(* Logix 5000 project; controller AdvManLab vendor 1 type 14 code 158 rev 28.12; software revision 28.01; part 12 of 13 *)
(* tags used below, declared in another part *)
   ABB_Loop_Conv_ES_Ch1 : BOOL;   // Cell 3 Conveyor Pull Cord / E-Stop Ch1
   ABB_Loop_Conv_ES_Ch2 : BOOL;   // Cell 3 Conveyor Pull Cord / E-Stop Ch2
   ABBLoopSTO_O1 : BOOL;
   ABBLoopSTO_O2 : BOOL;
   C1_Robot_ES_OK : BOOL;
   C1_Robot_Gates_OK : BOOL;
   C1EASRelay_Monitor : BOOL;   // Robot External Safety Gate Relay Monitor
   C1EESRelay_Monitor : BOOL;   // Robot External EStop Relay Monitor
   C1S : Fanuc_Cell_Safe;
   C2_Robot_ES_OK : BOOL;
   C2_Robot_Gates_OK : BOOL;
   C2EASRelay_Monitor : BOOL;   // Robot External Safety Gate Relay Monitor
   C2EESRelay_Monitor : BOOL;   // Robot External EStop Relay Monitor
   C2S : Fanuc_Cell_Safe;
   C3_Robot_ES_OK : BOOL;
   C3_Robot_Gates_OK : BOOL;
   C3EASRelay_Monitor : BOOL;   // Robot External Safety Gate Relay Monitor
   C3EESRelay_Monitor : BOOL;   // Robot External EStop Relay Monitor
   C3S : ABB_Cell_Safe;
   Cell_1 : Fanuc_Cell;
   Cell_2 : Fanuc_Cell;
   Fanuc_Loop_Conv_ES_Ch1 : BOOL;   // Cell 1/2 Conveyor Pull Cord / E-Stop Ch1
   Fanuc_Loop_Conv_ES_Ch2 : BOOL;   // Cell 1/2 Conveyor Pull Cord / E-Stop Ch2
   FanucLoopSTO_O1 : BOOL;
   FanucLoopSTO_O2 : BOOL;
   MainPnlESCH1 : BOOL;   // Main Panel E-Stop Button CH1
   MainPnlESCH2 : BOOL;   // Main Panel E-Stop Button CH2
   RungCommentS : BOOL;
   Unused_S_In : BOOL;   // Tag to indicate bit is unused in I/O mapping
   Unused_S_Out : BOOL;   // Unused Safety Output - Replace as needed
(* SafetyProgram, continued *)

ROUTINE MainRoutine   (* ladder *)
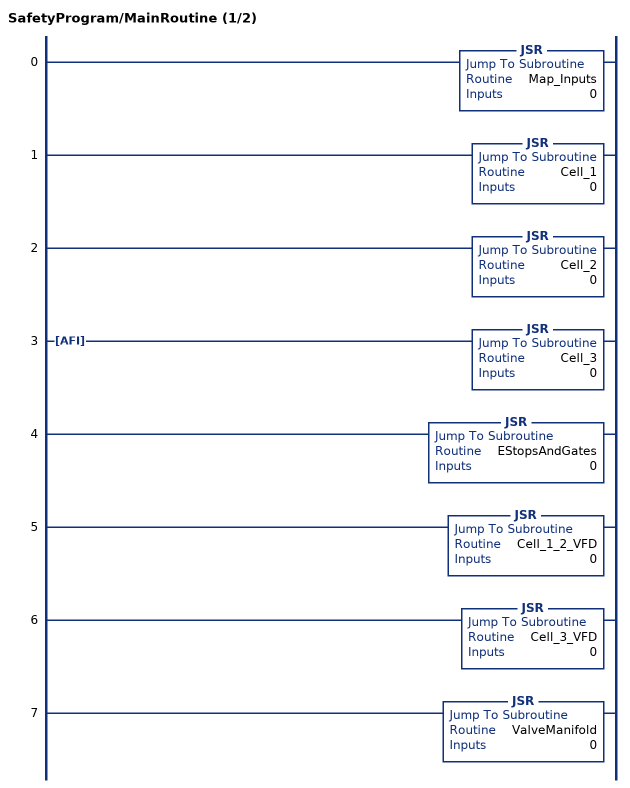
   0: JSR(Map_Inputs,0);
   1: JSR(Cell_1,0);
   2: JSR(Cell_2,0);
   3: AFI()JSR(Cell_3,0);
   4: JSR(EStopsAndGates,0);
   5: JSR(Cell_1_2_VFD,0);
   6: JSR(Cell_3_VFD,0);
   7: JSR(ValveManifold,0);
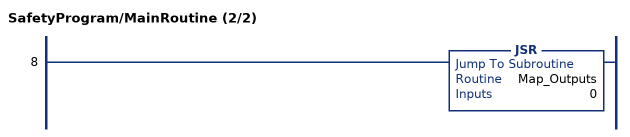
   8: JSR(Map_Outputs,0);
END_ROUTINE

ROUTINE Map_Inputs   (* ladder *)
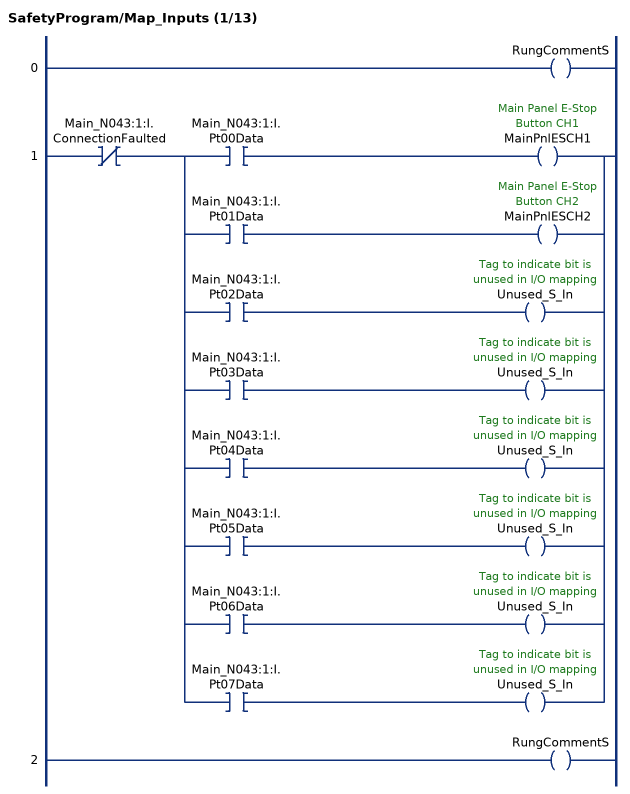
   0: OTE(RungCommentS);
   1: XIO(Main_N043:1:I.ConnectionFaulted)[XIC(Main_N043:1:I.Pt00Data) OTE(MainPnlESCH1) ,XIC(Main_N043:1:I.Pt01Data) OTE(MainPnlESCH2) ,XIC(Main_N043:1:I.Pt02Data) OTE(Unused_S_In) ,XIC(Main_N043:1:I.Pt03Data) OTE(Unused_S_In) ,XIC(Main_N043:1:I.Pt04Data) OTE(Unused_S_In) ,XIC(Main_N043:1:I.Pt05Data) OTE(Unused_S_In) ,XIC(Main_N043:1:I.Pt06Data) OTE(Unused_S_In) ,XIC(Main_N043:1:I.Pt07Data) OTE(Unused_S_In) ];
   2: OTE(RungCommentS);
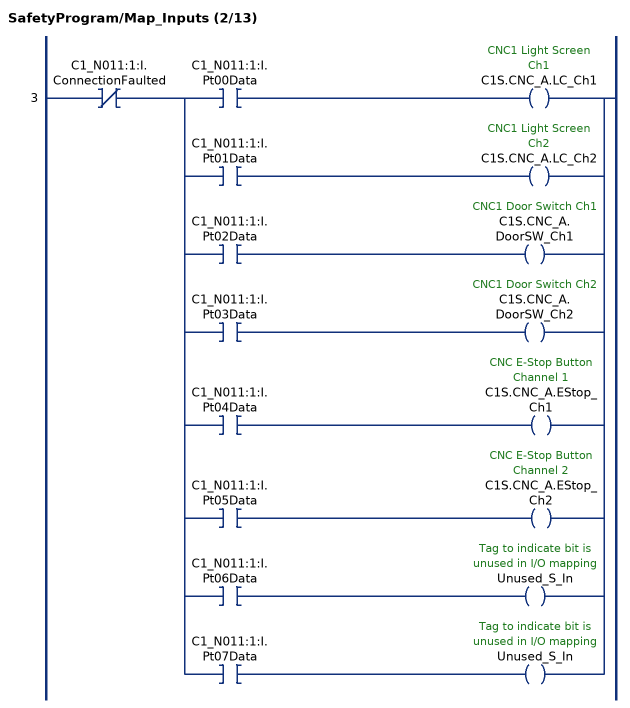
   3: XIO(C1_N011:1:I.ConnectionFaulted)[XIC(C1_N011:1:I.Pt00Data) OTE(C1S.CNC_A.LC_Ch1) ,XIC(C1_N011:1:I.Pt01Data) OTE(C1S.CNC_A.LC_Ch2) ,XIC(C1_N011:1:I.Pt02Data) OTE(C1S.CNC_A.DoorSW_Ch1) ,XIC(C1_N011:1:I.Pt03Data) OTE(C1S.CNC_A.DoorSW_Ch2) ,XIC(C1_N011:1:I.Pt04Data) OTE(C1S.CNC_A.EStop_Ch1) ,XIC(C1_N011:1:I.Pt05Data) OTE(C1S.CNC_A.EStop_Ch2) ,XIC(C1_N011:1:I.Pt06Data) OTE(Unused_S_In) ,XIC(C1_N011:1:I.Pt07Data) OTE(Unused_S_In) ];
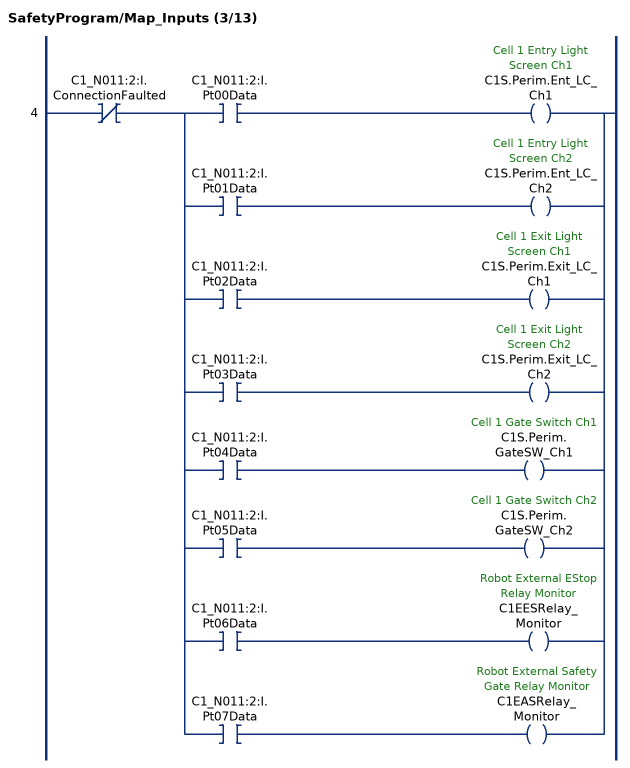
   4: XIO(C1_N011:2:I.ConnectionFaulted)[XIC(C1_N011:2:I.Pt00Data) OTE(C1S.Perim.Ent_LC_Ch1) ,XIC(C1_N011:2:I.Pt01Data) OTE(C1S.Perim.Ent_LC_Ch2) ,XIC(C1_N011:2:I.Pt02Data) OTE(C1S.Perim.Exit_LC_Ch1) ,XIC(C1_N011:2:I.Pt03Data) OTE(C1S.Perim.Exit_LC_Ch2) ,XIC(C1_N011:2:I.Pt04Data) OTE(C1S.Perim.GateSW_Ch1) ,XIC(C1_N011:2:I.Pt05Data) OTE(C1S.Perim.GateSW_Ch2) ,XIC(C1_N011:2:I.Pt06Data) OTE(C1EESRelay_Monitor) ,XIC(C1_N011:2:I.Pt07Data) OTE(C1EASRelay_Monitor) ];
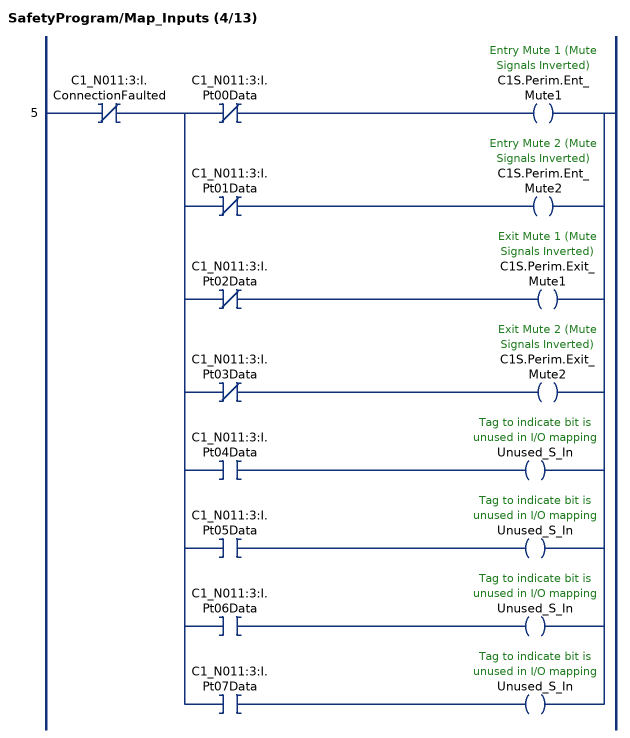
   5: XIO(C1_N011:3:I.ConnectionFaulted)[XIO(C1_N011:3:I.Pt00Data) OTE(C1S.Perim.Ent_Mute1) ,XIO(C1_N011:3:I.Pt01Data) OTE(C1S.Perim.Ent_Mute2) ,XIO(C1_N011:3:I.Pt02Data) OTE(C1S.Perim.Exit_Mute1) ,XIO(C1_N011:3:I.Pt03Data) OTE(C1S.Perim.Exit_Mute2) ,XIC(C1_N011:3:I.Pt04Data) OTE(Unused_S_In) ,XIC(C1_N011:3:I.Pt05Data) OTE(Unused_S_In) ,XIC(C1_N011:3:I.Pt06Data) OTE(Unused_S_In) ,XIC(C1_N011:3:I.Pt07Data) OTE(Unused_S_In) ];
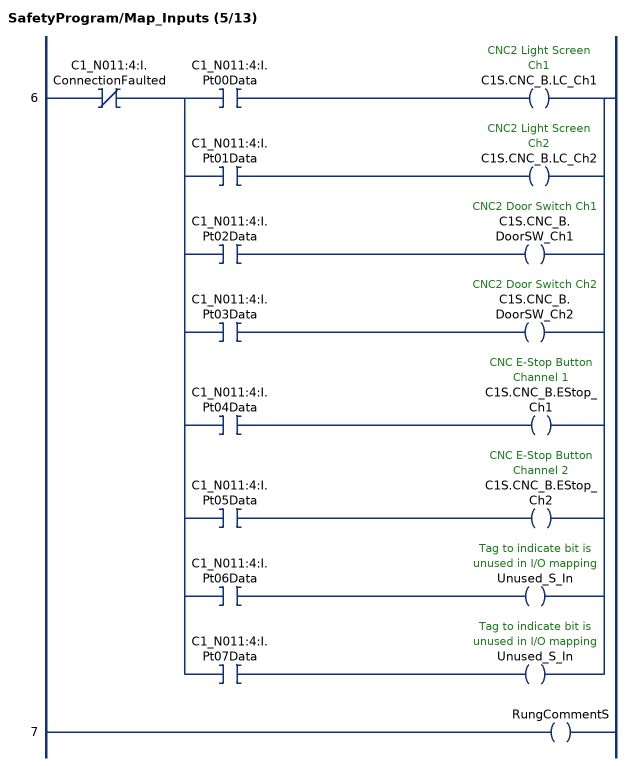
   6: XIO(C1_N011:4:I.ConnectionFaulted)[XIC(C1_N011:4:I.Pt00Data) OTE(C1S.CNC_B.LC_Ch1) ,XIC(C1_N011:4:I.Pt01Data) OTE(C1S.CNC_B.LC_Ch2) ,XIC(C1_N011:4:I.Pt02Data) OTE(C1S.CNC_B.DoorSW_Ch1) ,XIC(C1_N011:4:I.Pt03Data) OTE(C1S.CNC_B.DoorSW_Ch2) ,XIC(C1_N011:4:I.Pt04Data) OTE(C1S.CNC_B.EStop_Ch1) ,XIC(C1_N011:4:I.Pt05Data) OTE(C1S.CNC_B.EStop_Ch2) ,XIC(C1_N011:4:I.Pt06Data) OTE(Unused_S_In) ,XIC(C1_N011:4:I.Pt07Data) OTE(Unused_S_In) ];
   7: OTE(RungCommentS);
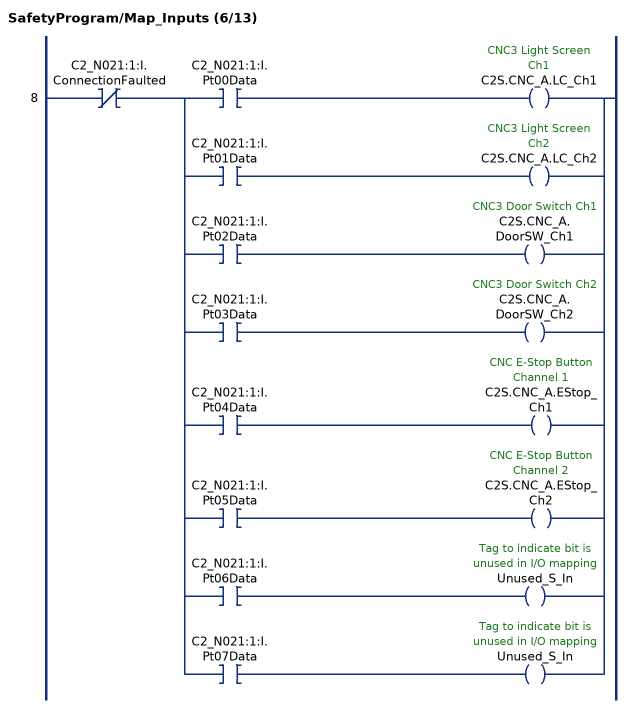
   8: XIO(C2_N021:1:I.ConnectionFaulted)[XIC(C2_N021:1:I.Pt00Data) OTE(C2S.CNC_A.LC_Ch1) ,XIC(C2_N021:1:I.Pt01Data) OTE(C2S.CNC_A.LC_Ch2) ,XIC(C2_N021:1:I.Pt02Data) OTE(C2S.CNC_A.DoorSW_Ch1) ,XIC(C2_N021:1:I.Pt03Data) OTE(C2S.CNC_A.DoorSW_Ch2) ,XIC(C2_N021:1:I.Pt04Data) OTE(C2S.CNC_A.EStop_Ch1) ,XIC(C2_N021:1:I.Pt05Data) OTE(C2S.CNC_A.EStop_Ch2) ,XIC(C2_N021:1:I.Pt06Data) OTE(Unused_S_In) ,XIC(C2_N021:1:I.Pt07Data) OTE(Unused_S_In) ];
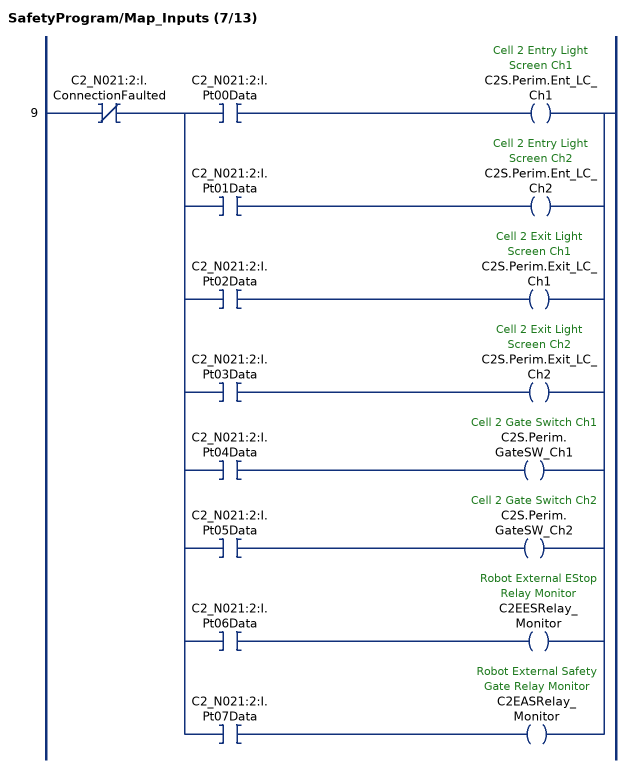
   9: XIO(C2_N021:2:I.ConnectionFaulted)[XIC(C2_N021:2:I.Pt00Data) OTE(C2S.Perim.Ent_LC_Ch1) ,XIC(C2_N021:2:I.Pt01Data) OTE(C2S.Perim.Ent_LC_Ch2) ,XIC(C2_N021:2:I.Pt02Data) OTE(C2S.Perim.Exit_LC_Ch1) ,XIC(C2_N021:2:I.Pt03Data) OTE(C2S.Perim.Exit_LC_Ch2) ,XIC(C2_N021:2:I.Pt04Data) OTE(C2S.Perim.GateSW_Ch1) ,XIC(C2_N021:2:I.Pt05Data) OTE(C2S.Perim.GateSW_Ch2) ,XIC(C2_N021:2:I.Pt06Data) OTE(C2EESRelay_Monitor) ,XIC(C2_N021:2:I.Pt07Data) OTE(C2EASRelay_Monitor) ];
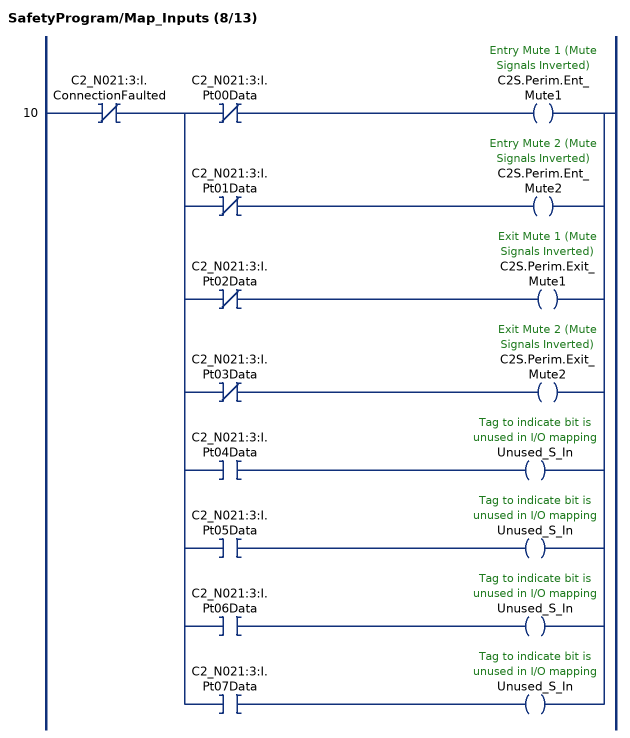
   10: XIO(C2_N021:3:I.ConnectionFaulted)[XIO(C2_N021:3:I.Pt00Data) OTE(C2S.Perim.Ent_Mute1) ,XIO(C2_N021:3:I.Pt01Data) OTE(C2S.Perim.Ent_Mute2) ,XIO(C2_N021:3:I.Pt02Data) OTE(C2S.Perim.Exit_Mute1) ,XIO(C2_N021:3:I.Pt03Data) OTE(C2S.Perim.Exit_Mute2) ,XIC(C2_N021:3:I.Pt04Data) OTE(Unused_S_In) ,XIC(C2_N021:3:I.Pt05Data) OTE(Unused_S_In) ,XIC(C2_N021:3:I.Pt06Data) OTE(Unused_S_In) ,XIC(C2_N021:3:I.Pt07Data) OTE(Unused_S_In) ];
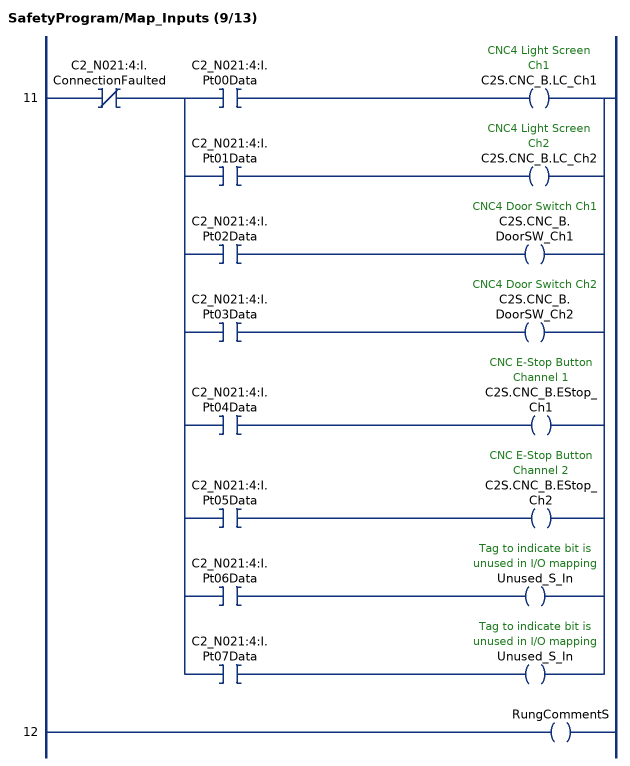
   11: XIO(C2_N021:4:I.ConnectionFaulted)[XIC(C2_N021:4:I.Pt00Data) OTE(C2S.CNC_B.LC_Ch1) ,XIC(C2_N021:4:I.Pt01Data) OTE(C2S.CNC_B.LC_Ch2) ,XIC(C2_N021:4:I.Pt02Data) OTE(C2S.CNC_B.DoorSW_Ch1) ,XIC(C2_N021:4:I.Pt03Data) OTE(C2S.CNC_B.DoorSW_Ch2) ,XIC(C2_N021:4:I.Pt04Data) OTE(C2S.CNC_B.EStop_Ch1) ,XIC(C2_N021:4:I.Pt05Data) OTE(C2S.CNC_B.EStop_Ch2) ,XIC(C2_N021:4:I.Pt06Data) OTE(Unused_S_In) ,XIC(C2_N021:4:I.Pt07Data) OTE(Unused_S_In) ];
   12: OTE(RungCommentS);
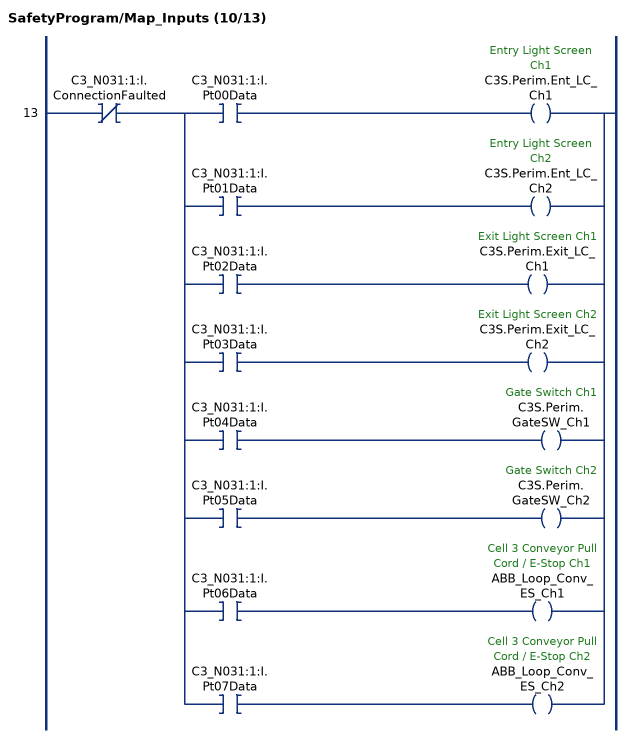
   13: XIO(C3_N031:1:I.ConnectionFaulted)[XIC(C3_N031:1:I.Pt00Data) OTE(C3S.Perim.Ent_LC_Ch1) ,XIC(C3_N031:1:I.Pt01Data) OTE(C3S.Perim.Ent_LC_Ch2) ,XIC(C3_N031:1:I.Pt02Data) OTE(C3S.Perim.Exit_LC_Ch1) ,XIC(C3_N031:1:I.Pt03Data) OTE(C3S.Perim.Exit_LC_Ch2) ,XIC(C3_N031:1:I.Pt04Data) OTE(C3S.Perim.GateSW_Ch1) ,XIC(C3_N031:1:I.Pt05Data) OTE(C3S.Perim.GateSW_Ch2) ,XIC(C3_N031:1:I.Pt06Data) OTE(ABB_Loop_Conv_ES_Ch1) ,XIC(C3_N031:1:I.Pt07Data) OTE(ABB_Loop_Conv_ES_Ch2) ];
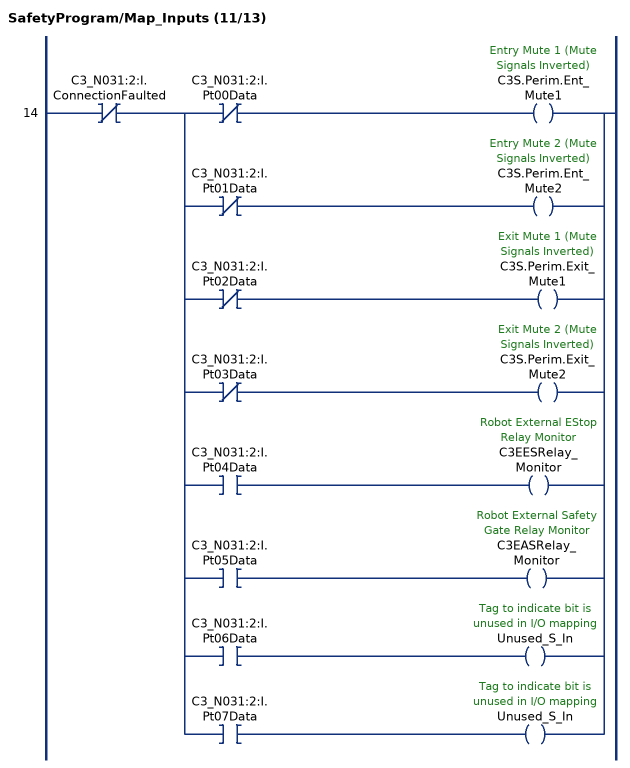
   14: XIO(C3_N031:2:I.ConnectionFaulted)[XIO(C3_N031:2:I.Pt00Data) OTE(C3S.Perim.Ent_Mute1) ,XIO(C3_N031:2:I.Pt01Data) OTE(C3S.Perim.Ent_Mute2) ,XIO(C3_N031:2:I.Pt02Data) OTE(C3S.Perim.Exit_Mute1) ,XIO(C3_N031:2:I.Pt03Data) OTE(C3S.Perim.Exit_Mute2) ,XIC(C3_N031:2:I.Pt04Data) OTE(C3EESRelay_Monitor) ,XIC(C3_N031:2:I.Pt05Data) OTE(C3EASRelay_Monitor) ,XIC(C3_N031:2:I.Pt06Data) OTE(Unused_S_In) ,XIC(C3_N031:2:I.Pt07Data) OTE(Unused_S_In) ];
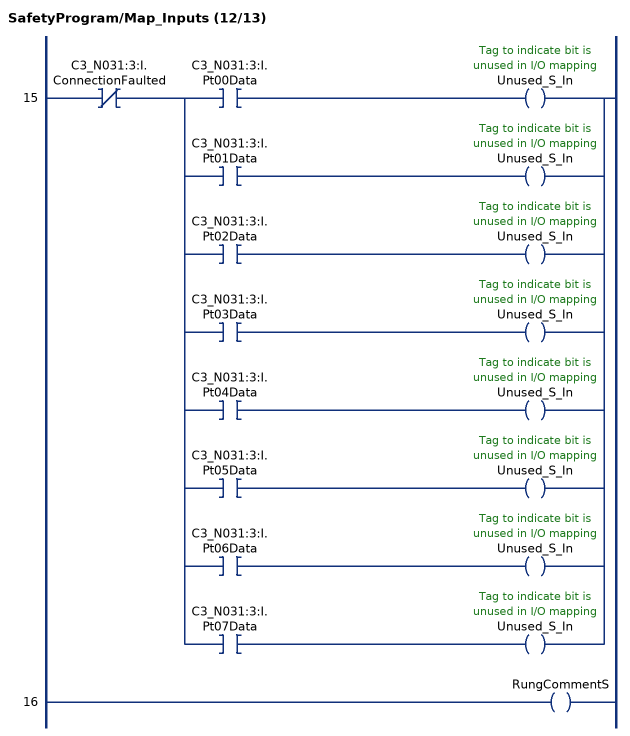
   15: XIO(C3_N031:3:I.ConnectionFaulted)[XIC(C3_N031:3:I.Pt00Data) OTE(Unused_S_In) ,XIC(C3_N031:3:I.Pt01Data) OTE(Unused_S_In) ,XIC(C3_N031:3:I.Pt02Data) OTE(Unused_S_In) ,XIC(C3_N031:3:I.Pt03Data) OTE(Unused_S_In) ,XIC(C3_N031:3:I.Pt04Data) OTE(Unused_S_In) ,XIC(C3_N031:3:I.Pt05Data) OTE(Unused_S_In) ,XIC(C3_N031:3:I.Pt06Data) OTE(Unused_S_In) ,XIC(C3_N031:3:I.Pt07Data) OTE(Unused_S_In) ];
   16: OTE(RungCommentS);
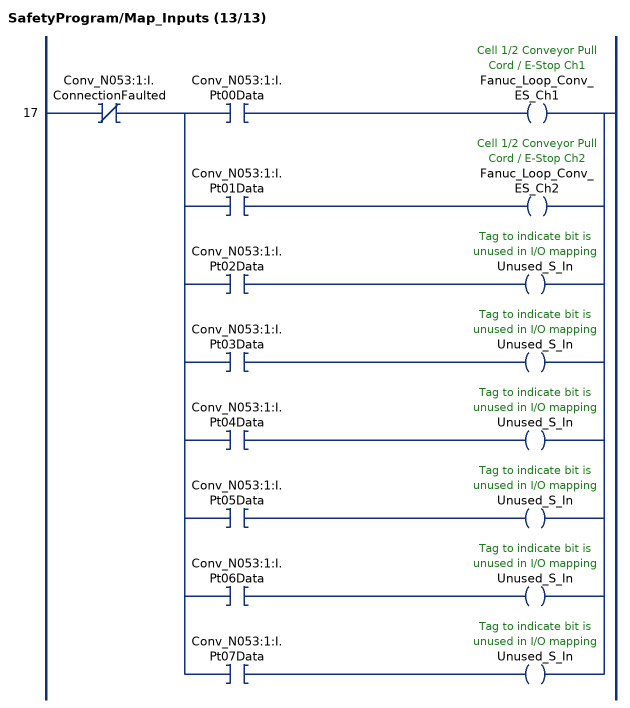
   17: XIO(Conv_N053:1:I.ConnectionFaulted)[XIC(Conv_N053:1:I.Pt00Data) OTE(Fanuc_Loop_Conv_ES_Ch1) ,XIC(Conv_N053:1:I.Pt01Data) OTE(Fanuc_Loop_Conv_ES_Ch2) ,XIC(Conv_N053:1:I.Pt02Data) OTE(Unused_S_In) ,XIC(Conv_N053:1:I.Pt03Data) OTE(Unused_S_In) ,XIC(Conv_N053:1:I.Pt04Data) OTE(Unused_S_In) ,XIC(Conv_N053:1:I.Pt05Data) OTE(Unused_S_In) ,XIC(Conv_N053:1:I.Pt06Data) OTE(Unused_S_In) ,XIC(Conv_N053:1:I.Pt07Data) OTE(Unused_S_In) ];
END_ROUTINE

ROUTINE Map_Outputs   (* ladder *)
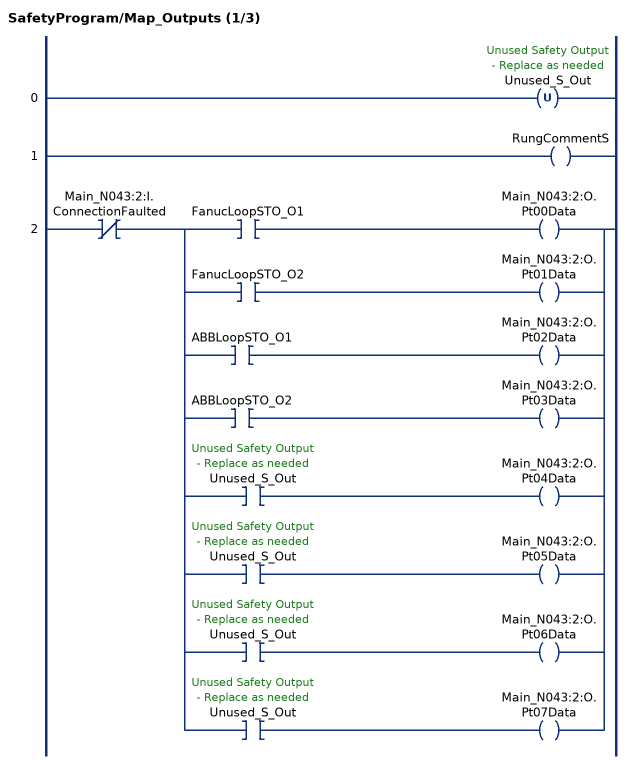
   0: OTU(Unused_S_Out);
   1: OTE(RungCommentS);
   2: XIO(Main_N043:2:I.ConnectionFaulted)[XIC(FanucLoopSTO_O1) OTE(Main_N043:2:O.Pt00Data) ,XIC(FanucLoopSTO_O2) OTE(Main_N043:2:O.Pt01Data) ,XIC(ABBLoopSTO_O1) OTE(Main_N043:2:O.Pt02Data) ,XIC(ABBLoopSTO_O2) OTE(Main_N043:2:O.Pt03Data) ,XIC(Unused_S_Out) OTE(Main_N043:2:O.Pt04Data) ,XIC(Unused_S_Out) OTE(Main_N043:2:O.Pt05Data) ,XIC(Unused_S_Out) OTE(Main_N043:2:O.Pt06Data) ,XIC(Unused_S_Out) OTE(Main_N043:2:O.Pt07Data) ];
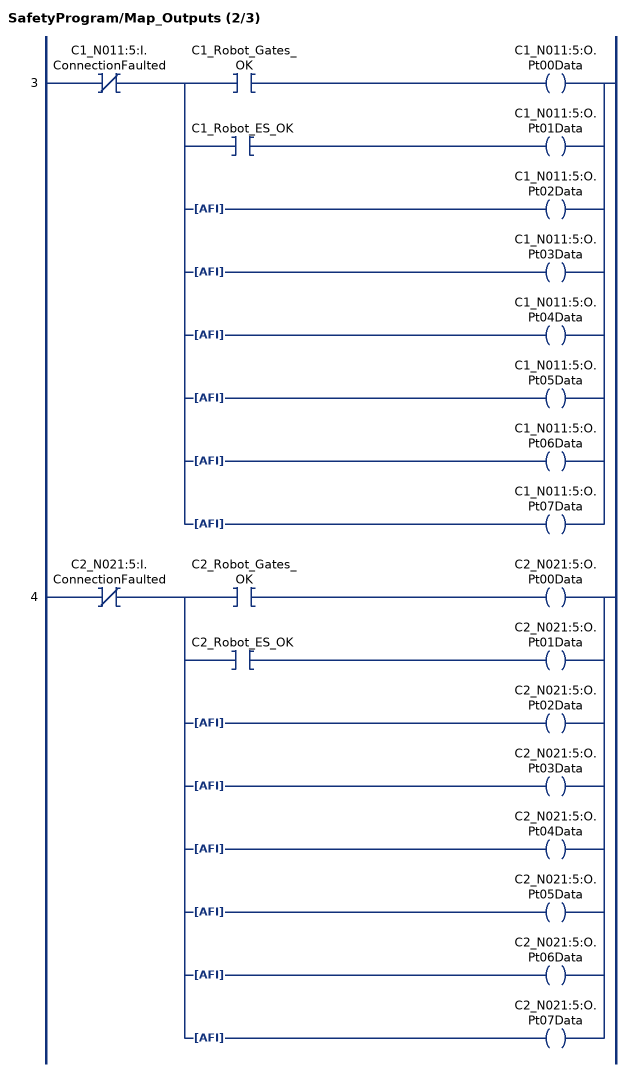
   3: XIO(C1_N011:5:I.ConnectionFaulted)[XIC(C1_Robot_Gates_OK) OTE(C1_N011:5:O.Pt00Data) ,XIC(C1_Robot_ES_OK) OTE(C1_N011:5:O.Pt01Data) ,AFI() OTE(C1_N011:5:O.Pt02Data) ,AFI() OTE(C1_N011:5:O.Pt03Data) ,AFI() OTE(C1_N011:5:O.Pt04Data) ,AFI() OTE(C1_N011:5:O.Pt05Data) ,AFI() OTE(C1_N011:5:O.Pt06Data) ,AFI() OTE(C1_N011:5:O.Pt07Data) ];
   4: XIO(C2_N021:5:I.ConnectionFaulted)[XIC(C2_Robot_Gates_OK) OTE(C2_N021:5:O.Pt00Data) ,XIC(C2_Robot_ES_OK) OTE(C2_N021:5:O.Pt01Data) ,AFI() OTE(C2_N021:5:O.Pt02Data) ,AFI() OTE(C2_N021:5:O.Pt03Data) ,AFI() OTE(C2_N021:5:O.Pt04Data) ,AFI() OTE(C2_N021:5:O.Pt05Data) ,AFI() OTE(C2_N021:5:O.Pt06Data) ,AFI() OTE(C2_N021:5:O.Pt07Data) ];
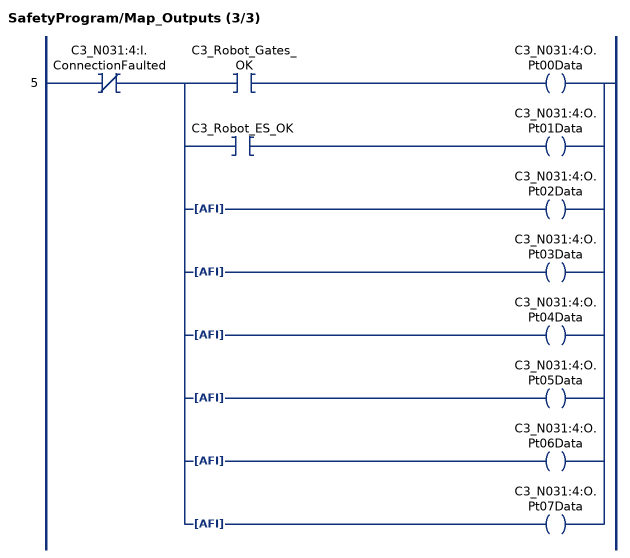
   5: XIO(C3_N031:4:I.ConnectionFaulted)[XIC(C3_Robot_Gates_OK) OTE(C3_N031:4:O.Pt00Data) ,XIC(C3_Robot_ES_OK) OTE(C3_N031:4:O.Pt01Data) ,AFI() OTE(C3_N031:4:O.Pt02Data) ,AFI() OTE(C3_N031:4:O.Pt03Data) ,AFI() OTE(C3_N031:4:O.Pt04Data) ,AFI() OTE(C3_N031:4:O.Pt05Data) ,AFI() OTE(C3_N031:4:O.Pt06Data) ,AFI() OTE(C3_N031:4:O.Pt07Data) ];
END_ROUTINE
